Staubli VAL3: socketWrite.pgx

program socketWrite(string& sBuffer (dimensions=1), num& nBuffer[] (dimensions=1))
  local num ni
begin
  if len(sBuffer)>29
    sBuffer=left(sBuffer,29)
  endIf
  for ni=0 to 29 step 1
    nBuffer[ni]=0
  endFor
  for ni=0 to (len(sBuffer)-1) step 1
    nBuffer[ni]=asc(sBuffer,ni)
  endFor
  nBuffer[ni]=13
end
